// TIA Portal project "Garaje" (V16)

(* hardware
DEVICE "S7-1200 station_2"  S7-1200 Station
   slot 0: "Rack_0"  S7-1200 Rack  Rack  V1.0
   slot 1: "PLC_2"  CPU 1214C AC/DC/Rly  6ES7 214-1BG40-0XB0  V4.2
   slot 3: "AQ 1x12BIT_1"  AQ1 signal board  6ES7 232-4HA30-0XB0  V1.0
*)

// ===== PLC "PLC_2"  CPU 1214C AC/DC/Rly =====

VAR_GLOBAL   // PLC tag table "Estados"
   "estado0" AT %M0.0 : Bool;
   "estado1" AT %M0.1 : Bool;
   "estado2" AT %M0.2 : Bool;
   "estado3" AT %M0.3 : Bool;
END_VAR

VAR_GLOBAL   // PLC tag table "Entradas"
   "timer" AT %I0.7 : Bool;
   "mando" AT %I0.0 : Bool;
   "fcArriba" AT %I0.1 : Bool;
   "fcAbajo" AT %I0.2 : Bool;
   "cFotoelec" AT %I0.3 : Bool;
END_VAR

VAR_GLOBAL   // PLC tag table "Salidas"
   "motor¡" AT %Q0.0 : Bool;
   "motor!" AT %Q0.1 : Bool;
END_VAR

// folder: System blocks/Program resources

DATA_BLOCK "Timer_10s"   // DB1
{ S7_Optimized_Access := 'TRUE' }
AUTHOR : Simatic
FAMILY : IEC
NAME : IEC_TMR
VERSION : 1.0
// stored: InstanceOfName IEC_TIMER
"IEC_TIMER"
BEGIN
END_DATA_BLOCK

// folder: (top level)

ORGANIZATION_BLOCK "Main"   // OB1, LAD, ProgramCycle
TITLE = "Main Program Sweep (Cycle)"
{ S7_Optimized_Access := 'TRUE' }
VERSION : 0.1
   VAR_INPUT
      Initial_Call : Bool;   // Initial call of this OB
      Remanence : Bool;   // =True, if remanent data are available
   END_VAR
BEGIN

REGION Network 1: Temporizadores
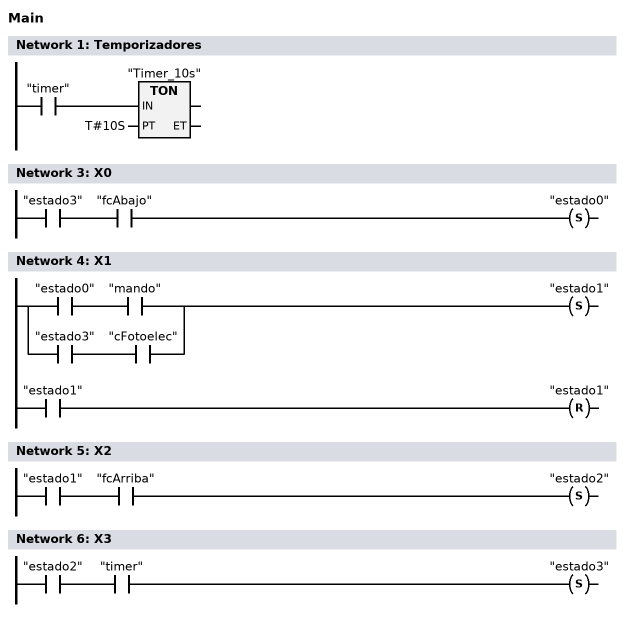
   "Timer_10s".TON(IN := "timer", PT := T#10S);
END_REGION

REGION Network 2 (SCL): X2
   // en SCL
END_REGION

REGION Network 3: X0
   RUNG wire#powerrail
      Contact( "estado3" )
      Contact( "fcAbajo" )
      S_Coil( "estado0" )
   END_RUNG
   // the same network as SCL:
   IF "estado3" AND "fcAbajo" THEN "estado0" := TRUE; END_IF;
END_REGION

REGION Network 4: X1
   RUNG wire#powerrail
      Contact( "estado0" )
      Contact( "mando" )
      wire#w1
      S_Coil( "estado1" )
   END_RUNG
   RUNG wire#powerrail
      Contact( "estado3" )
      Contact( "cFotoelec" )
   END_RUNG wire#w1
   RUNG wire#powerrail
      Contact( "estado1" )
      R_Coil( "estado1" )
   END_RUNG
   // the same network as SCL:
   IF ("estado0" AND "mando") OR ("estado3" AND "cFotoelec") THEN "estado1" := TRUE; END_IF;
   IF "estado1" THEN "estado1" := FALSE; END_IF;
END_REGION

REGION Network 5: X2
   RUNG wire#powerrail
      Contact( "estado1" )
      Contact( "fcArriba" )
      S_Coil( "estado2" )
   END_RUNG
   // the same network as SCL:
   IF "estado1" AND "fcArriba" THEN "estado2" := TRUE; END_IF;
END_REGION

REGION Network 6: X3
   RUNG wire#powerrail
      Contact( "estado2" )
      Contact( "timer" )
      S_Coil( "estado3" )
   END_RUNG
   // the same network as SCL:
   IF "estado2" AND "timer" THEN "estado3" := TRUE; END_IF;
END_REGION

REGION Network 7: X3
   // FUNCTION BLOCK DIAGRAM
END_REGION
END_ORGANIZATION_BLOCK